FUNCTION_BLOCK FB_PIZZA_OVEN

VAR_INPUT
	btn_PutAPizza:BOOL;
	btn_PackageThePizza:BOOL;
	bReset:BOOL;
	iFlavor:INT;
	iTime4Cooking:DINT:=1;
END_VAR


VAR_OUTPUT
		iTotalPizzasCooked :UDINT;
		iTotalPizzasBurned :UDINT;
		InpCookingTime:DINT;
		sCookingTime :DINT;
		LightCooking:BOOL;
 		LBuzzer:BOOL;
		sStateDescription :STRING;
		sPizzaDescription :STRING;
		sPizzaDescription2 :STRING;
END_VAR


VAR
	fbMyTimer : TON; //timer
	iState : DINT;
	bs_PizzaOnEntrit : BOOL;
	bs_PizzaOnOven : BOOL;
	bs_PizzaOnExit : BOOL;
	bBurnt :BOOL;
	bBurnt2 :BOOL;
	tTime4Cooking:TIME;
	bFlavor1:BOOL:=FALSE;
	bFlavor2:BOOL:=FALSE;
	bFlavor3:BOOL:=FALSE;
END_VAR

tTime4Cooking:=DINT_TO_TIME(iTime4Cooking*1000);

IF btn_PutAPizza THEN
	bs_PizzaOnEntrit:=TRUE;
	IF int_to_bool(iFlavor) THEN
		bFlavor1:=TRUE;
	ELSE
		bFlavor1:=FALSE;	
	END_IF
END_IF

IF btn_PackageThePizza THEN
	bs_PizzaOnExit:=FALSE;
	bFlavor3:=FALSE;
END_IF

IF bReset THEN
	bReset:=FALSE;
	iTotalPizzasCooked:=0;
	iTotalPizzasBurned:=0;
END_IF


CASE iState OF

	0: //wait for raw pizza 
		
		sStateDescription:='Waiting for pizza';
		IF bs_PizzaOnEntrit THEN
			IF bs_PizzaOnOven=FALSE THEN
				iState:=1;	
			END_IF
		END_IF
		
	1: //moving pizza
	
		sStateDescription:='Moving pizza';
		fbMyTimer(IN := TRUE,PT:=T#1S);
		IF fbMyTimer.Q THEN
			bs_PizzaOnOven:=TRUE;
			fbMyTimer(IN := FALSE);
			iState:=10;
			bs_PizzaOnEntrit:=FALSE;
			IF bFlavor1 THEN
				bFlavor2:=TRUE;
				bFlavor1:=FALSE;
			END_IF
		END_IF
		
	10: //there is a pizza, cook it
		
		sStateDescription:='Baking pizza';
		sPizzaDescription:='cooking';
		bBurnt:=false;
		LightCooking:=TRUE;
		sCookingTime:=(TIME_TO_DINT(fbMyTImer.ET))/1000;
		fbMyTimer(IN := TRUE,PT:=tTime4Cooking);
		IF fbMyTimer.Q THEN
			fbMyTimer(IN := FALSE);
			if bs_PizzaOnExit then
				iState:=20;
			else
				iState:=21;
			END_IF
			LightCooking:=FALSE;
			sCookingTime:=0;
		END_IF
		
	20: //burning pizza
	
		sStateDescription:='Pizza done, burning';
		sPizzaDescription:='burning';
		bBurnt:=true;
		IF NOT bs_PizzaOnExit THEN
			//simulating a conveyor
			bs_PizzaOnOven:=FALSE;
			bs_PizzaOnExit:=TRUE;
			IF bFlavor2 THEN
				bFlavor3:=TRUE;
				bFlavor2:=FALSE;
			END_IF
			iTotalPizzasBurned := iTotalPizzasBurned + 1;
			iState:=30;
			LBuzzer:=FALSE;
			sPizzaDescription2:='burned';
			bBurnt2:=TRUE;
		ELSE
			LBuzzer:=TRUE;
		END_IF
		
	21: //not burned pizza
	    sPizzaDescription2:='cooked';
		bBurnt2:=FALSE;
		iState:=30;
		bs_PizzaOnOven:=FALSE;
		bs_PizzaOnExit:=TRUE;
		IF bFlavor2 THEN
			bFlavor3:=TRUE;
			bFlavor2:=FALSE;
		END_IF
		iTotalPizzasCooked := iTotalPizzasCooked + 1;
		iState:=30;
		LBuzzer:=FALSE;
	
	30: //pizza just removed on output tray
	
		sStateDescription:='Please pack the pizza!';
		iState:=0; //wait for another pizza
		
END_CASE

END_FUNCTION_BLOCK

(* stored: Version 1.1.0.1, ProductVersion 3.1.4024.3
   POU FB_PIZZA_OVEN: Id {e6090a63-31f8-419b-84f0-8cedd9cd2065}, SpecialFunc None *)
